(* CODESYS project SPT_NC_Basic_Slave.library
   Company: Beckhoff Automation LLC
   DefaultNamespace: SPT_NCBasicSlave
   Version: 3.0.0
   Placeholder: SPT NC Basic Slave
   Title: SPT NC Basic Slave

Project tree, tasks and I/O mapping:
  libraries: SPT Base Types, * (Beckhoff Automation LLC); SPT NC Axis, * (Beckhoff Automation LLC); SPT NC Homing, * (Beckhoff Automation LLC); Tc2_MC2, * (Beckhoff Automation GmbH); Tc3_Module, * (Beckhoff Automation GmbH); Tc3_System, * (Beckhoff Automation GmbH)
  Function Blocks/
    function block FB_BasicSlaveAxis [ST]: Home, MoveAbsolute, MoveModulo, MoveRelative, MoveVelocity, Reset, GearIn, GearOut, InGear, Master1, Master2, Master3, Master4, RatioMaster1, RatioMaster2, RatioMaster3, RatioMaster4, Stop, CyclicLogic, CallFBs, Initialize
  Interfaces/
    interface I_BasicSlaveAxis: GearIn, GearOut, InGear, Master1, Master2, Master3, Master4, RatioMaster1, RatioMaster2, RatioMaster3, RatioMaster4
  Project Information/
    function F_GetCompany [ST]
    function F_GetTitle [ST]
    function F_GetVersion [ST]
  Version/
    global variables Global_Version
*)

// Version/Global_Version
{attribute 'TcGenerated'}
{attribute 'no-analysis'}
{attribute 'linkalways'}
// This function has been automatically generated from the project information.
VAR_GLOBAL CONSTANT
	{attribute 'const_non_replaced'}
	stLibVersion_SPT_NC_Basic_Slave : ST_LibVersion := (iMajor := 3, iMinor := 0, iBuild := 0, iRevision := 0, nFlags := 1, sVersion := '3.0.0');
END_VAR

// Function Blocks/FB_BasicSlaveAxis
FUNCTION_BLOCK FB_BasicSlaveAxis EXTENDS FB_BasicAxis IMPLEMENTS I_BasicSlaveAxis
VAR
    MCGearInMultimaster : MC_GearInMultiMaster;
    MCGearOut           : MC_GearOut;
    {attribute 'hide'}
    DummyAxis     : AXIS_REF;
    _Master1      : REFERENCE TO AXIS_REF;
    _Master2      : REFERENCE TO AXIS_REF;
    _Master3      : REFERENCE TO AXIS_REF;
    _Master4      : REFERENCE TO AXIS_REF;
    _RatioMaster1 : LREAL := 1;
    _RatioMaster2 : LREAL := 1;
    _RatioMaster3 : LREAL := 1;
    _RatioMaster4 : LREAL := 1;
END_VAR

//There should be no code in the function block body

METHOD Home : BOOL
IF _Busy OR _Error OR _HomeMethod = 0 THEN
    RETURN;
END_IF

MCGearInMultimaster(Slave := _Axis, Enable := FALSE);
Home := SUPER^.Home();
END_METHOD

METHOD MoveAbsolute : BOOL
VAR_INPUT
    Position      : LREAL;
    AbortPrevious : BOOL;
END_VAR
IF _Error THEN
    RETURN;
ELSE
    IF (_Busy AND NOT AbortPrevious) THEN
        RETURN;
    END_IF
END_IF

MCGearInMultimaster(Slave := _Axis, Enable := FALSE);
MoveAbsolute := SUPER^.MoveAbsolute(Position, AbortPrevious);
END_METHOD

METHOD MoveModulo : BOOL
VAR_INPUT
    Position      : LREAL;
    Direction     : MC_Direction;
    AbortPrevious : BOOL;
END_VAR
IF _Error THEN
    RETURN;
ELSE
    IF (_Busy AND NOT AbortPrevious) THEN
        RETURN;
    END_IF
END_IF

MCGearInMultimaster(Slave := _Axis, Enable := FALSE);
MoveModulo := SUPER^.MoveModulo(Position, Direction, AbortPrevious);
END_METHOD

METHOD MoveRelative : BOOL
VAR_INPUT
    Distance      : LREAL;
    AbortPrevious : BOOL;
END_VAR
IF _Error THEN
    RETURN;
ELSE
    IF (_Busy AND NOT AbortPrevious) THEN
        RETURN;
    END_IF
END_IF

MCGearInMultimaster(Slave := _Axis, Enable := FALSE);
MoveRelative := SUPER^.MoveRelative(Distance, AbortPrevious);
END_METHOD

METHOD MoveVelocity : BOOL
VAR_INPUT
    Velocity      : LREAL;
    AbortPrevious : BOOL;
END_VAR
IF _Error THEN
    RETURN;
ELSE
    IF (_Busy AND NOT AbortPrevious) THEN
        RETURN;
    END_IF
END_IF

MCGearInMultimaster(Slave := _Axis, Enable := FALSE);
MoveVelocity := SUPER^.MoveVelocity(Velocity, AbortPrevious);
END_METHOD

METHOD Reset : BOOL
IF _Busy OR _Axis.Status.Coupled OR _ResetMethod = 0 THEN
    //If axis is coupled it should be reset through the master
    RETURN;
END_IF

IF _ResetMethod.Execute() THEN
    _Error   := FALSE;
    _ErrorID := 0;
    Reset    := TRUE;
END_IF
END_METHOD

METHOD PUBLIC GearIn : BOOL
VAR_INPUT
END_VAR
IF _Busy OR _Error THEN
    RETURN;
END_IF

MCGearInMultimaster(Master1      := _Master1,
                    Master2      := _Master2,
                    Master3      := _Master3,
                    Master4      := _Master4,
                    Slave        := _Axis,
                    Enable       := TRUE,
                    GearRatio1   := _RatioMaster1,
                    GearRatio2   := _RatioMaster2,
                    GearRatio3   := _RatioMaster3,
                    GearRatio4   := _RatioMaster4,
                    Acceleration := _Acceleration,
                    Deceleration := _Deceleration,
                    Jerk         := _Jerk);

GearIn := TRUE;
END_METHOD

METHOD GearOut : BOOL
IF _Busy THEN
    RETURN;
END_IF

MCGearInMultimaster(Master1      := _Master1,
                    Master2      := _Master2,
                    Master3      := _Master3,
                    Master4      := _Master4,
                    Slave        := _Axis,
                    Enable       := FALSE,
                    GearRatio1   := _RatioMaster1,
                    GearRatio2   := _RatioMaster2,
                    GearRatio3   := _RatioMaster3,
                    GearRatio4   := _RatioMaster4,
                    Acceleration := _Acceleration,
                    Deceleration := _Deceleration,
                    Jerk         := _Jerk);

MCGearOut(Slave := _Axis, Execute := TRUE);
GearOut := TRUE;
END_METHOD

PROPERTY InGear : BOOL
GET
InGear := MCGearInMultimaster.InGear;
END_GET
END_PROPERTY

PROPERTY Master1 : REFERENCE TO AXIS_REF
GET
IF __ISVALIDREF(_Master1) THEN
    Master1 REF= _Master1;
END_IF
END_GET
SET
_Master1 REF= Master1;
END_SET
END_PROPERTY

PROPERTY Master2 : REFERENCE TO AXIS_REF
GET
IF __ISVALIDREF(_Master2) THEN
    Master2 REF= _Master2;
END_IF
END_GET
SET
_Master2 REF= Master2;
END_SET
END_PROPERTY

PROPERTY Master3 : REFERENCE TO AXIS_REF
GET
IF __ISVALIDREF(_Master3) THEN
    Master3 REF= _Master3;
END_IF
END_GET
SET
_Master3 REF= Master3;
END_SET
END_PROPERTY

PROPERTY Master4 : REFERENCE TO AXIS_REF
GET
IF __ISVALIDREF(_Master4) THEN
    Master4 REF= _Master4;
END_IF
END_GET
SET
_Master4 REF= Master4;
END_SET
END_PROPERTY

PROPERTY RatioMaster1 : LREAL
GET
RatioMaster1 := _RatioMaster1;
END_GET
SET
IF RatioMaster1 <> 0 THEN
    _RatioMaster1 := RatioMaster1;
END_IF
END_SET
END_PROPERTY

PROPERTY RatioMaster2 : LREAL
GET
RatioMaster2 := _RatioMaster2;
END_GET
SET
IF RatioMaster2 <> 0 THEN
    _RatioMaster2 := RatioMaster2;
END_IF
END_SET
END_PROPERTY

PROPERTY RatioMaster3 : LREAL
GET
RatioMaster3 := _RatioMaster3;
END_GET
SET
IF RatioMaster3 <> 0 THEN
    _RatioMaster3 := RatioMaster3;
END_IF
END_SET
END_PROPERTY

PROPERTY RatioMaster4 : LREAL
GET
RatioMaster4 := _RatioMaster4;
END_GET
SET
IF RatioMaster4 <> 0 THEN
    _RatioMaster4 := RatioMaster4;
END_IF
END_SET
END_PROPERTY

METHOD Stop : BOOL
MCGearInMultimaster(Slave := _Axis, Enable := FALSE);
IF SUPER^.Stop() THEN
    Stop := TRUE;
END_IF
END_METHOD

METHOD PUBLIC CyclicLogic
VAR_INPUT
END_VAR
IF NOT _InitComplete THEN
    _InitComplete := THIS^.Initialize();
    RETURN;
END_IF

//Call local FBs
SUPER^.CyclicLogic();
END_METHOD

METHOD PROTECTED CallFBs : BOOL
VAR_INPUT
END_VAR
SUPER^.CallFBs();

(* MC_GearInMultimaster *)
MCGearInMultimaster(Slave        := _Axis,
                    GearRatio1   := _RatioMaster1,
                    GearRatio2   := _RatioMaster2,
                    GearRatio3   := _RatioMaster3,
                    GearRatio4   := _RatioMaster4,
                    Acceleration := _Acceleration,
                    Deceleration := _Deceleration,
                    Jerk         := _Jerk);

//IF NOT MCGearInMultimaster.Busy THEN
IF MCGearInMultimaster.Error THEN
    _Error   := TRUE;
    _ErrorID := MCGearInMultimaster.ErrorID;
END_IF

//	MCGearInMultimaster(Slave := _Axis,Enable:= FALSE);

//END_IF

(* MC_GearOut *)
MCGearOut(Slave := _Axis);
IF NOT MCGearOut.Busy THEN
    IF MCGearOut.Error THEN
        _Error   := TRUE;
        _ErrorID := MCGearOut.ErrorID;
    END_IF

    MCGearOut(Slave := _Axis, Execute := FALSE);
END_IF

_Busy := _Busy OR MCGearOut.Error;
END_METHOD

METHOD PROTECTED Initialize : BOOL
VAR_INPUT
END_VAR
_Master1   REF= DummyAxis;
_Master2   REF= DummyAxis;
_Master3   REF= DummyAxis;
_Master4   REF= DummyAxis;
Initialize := SUPER^.Initialize();
END_METHOD

END_FUNCTION_BLOCK

// Interfaces/I_BasicSlaveAxis
INTERFACE I_BasicSlaveAxis EXTENDS I_BasicAxis

METHOD PUBLIC GearIn : BOOL
VAR_INPUT
END_VAR
END_METHOD

METHOD GearOut : BOOL
END_METHOD

PROPERTY InGear : BOOL
GET
END_GET
END_PROPERTY

PROPERTY Master1 : REFERENCE TO AXIS_REF
GET
END_GET
SET
END_SET
END_PROPERTY

PROPERTY Master2 : REFERENCE TO AXIS_REF
GET
END_GET
SET
END_SET
END_PROPERTY

PROPERTY Master3 : REFERENCE TO AXIS_REF
GET
END_GET
SET
END_SET
END_PROPERTY

PROPERTY Master4 : REFERENCE TO AXIS_REF
GET
END_GET
SET
END_SET
END_PROPERTY

PROPERTY RatioMaster1 : LREAL
GET
END_GET
SET
END_SET
END_PROPERTY

PROPERTY RatioMaster2 : LREAL
GET
END_GET
SET
END_SET
END_PROPERTY

PROPERTY RatioMaster3 : LREAL
GET
END_GET
SET
END_SET
END_PROPERTY

PROPERTY RatioMaster4 : LREAL
GET
END_GET
SET
END_SET
END_PROPERTY

END_INTERFACE

// Project Information/F_GetCompany
// This function has been automatically generated from the project information.
{attribute 'signature_flag' := '1073741824'}
{attribute 'TcGenerated'}
{attribute 'no-analysis'}
FUNCTION F_GetCompany : WSTRING
VAR_INPUT
	
END_VAR

F_GetCompany := "Beckhoff Automation LLC";

END_FUNCTION

// Project Information/F_GetTitle
// This function has been automatically generated from the project information.
{attribute 'signature_flag' := '1073741824'}
{attribute 'TcGenerated'}
{attribute 'no-analysis'}
FUNCTION F_GetTitle : WSTRING
VAR_INPUT
	
END_VAR

F_GetTitle := "SPT NC Basic Slave";

END_FUNCTION

// Project Information/F_GetVersion
// This function has been automatically generated from the project information.
{attribute 'signature_flag' := '1073741824'}
{attribute 'TcGenerated'}
{attribute 'no-analysis'}
FUNCTION F_GetVersion : ST_LibVersion
VAR_INPUT
	
END_VAR

F_GetVersion.iMajor := 3;
F_GetVersion.iMinor := 0;
F_GetVersion.iBuild := 0;
F_GetVersion.iRevision := 0;
F_GetVersion.sVersion := '3.0.0';
F_GetVersion.nFlags := 1;

END_FUNCTION
